% RSLogix 500 project TRIPACK_J.RSS, saved by version 12.00.00.00 %
PROJECT "TRIPACK"    % processor: MicroLogix 1400 %

PROGRAM FILES
  LAD 2   92 rungs
  LAD 3   19 rungs
  LAD 4   43 rungs
  LAD 6   66 rungs
  LAD 18   72 rungs

DATA FILES
  O0 OUTPUT  15 elements
  I1 INPUT  12 elements
  S2 STATUS  66 elements
  B3 BINARY  50 elements
  T4 TIMER  45 elements
  C5 COUNTER  13 elements
  R6 CONTROL  1 elements
  N7 INTEGER  256 elements
  F8 FLOAT  64 elements
  N9   96 elements
  L11   51 elements
  RIX13   13 elements
  RIX14   13 elements
  T15   48 elements
  ST16   18 elements
  RIX17   14 elements
  MG19   11 elements
  MG20   14 elements
  MG22   21 elements

LADDER 2
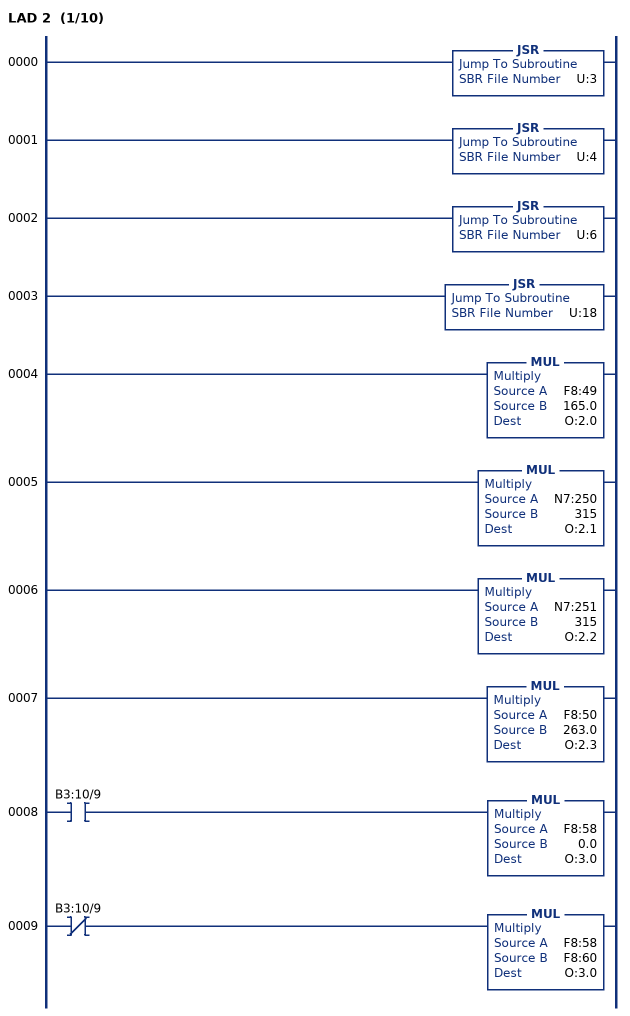
% Rung: 0 %
SOR JSR U:3 EOR
% Rung: 1 %
SOR JSR U:4 EOR
% Rung: 2 %
SOR JSR U:6 EOR
% Rung: 3 %
SOR JSR U:18 EOR
% Rung: 4 %
SOR MUL F8:49 165.0 O:2.0 EOR
% Rung: 5 %
SOR MUL N7:250 315 O:2.1 EOR
% Rung: 6 %
SOR MUL N7:251 315 O:2.2 EOR
% Rung: 7 %
SOR MUL F8:50 263.0 O:2.3 EOR
% Rung: 8 %
SOR XIC B3:10/9 MUL F8:58 0.0 O:3.0 EOR
% Rung: 9 %
SOR XIO B3:10/9 MUL F8:58 F8:60 O:3.0 EOR

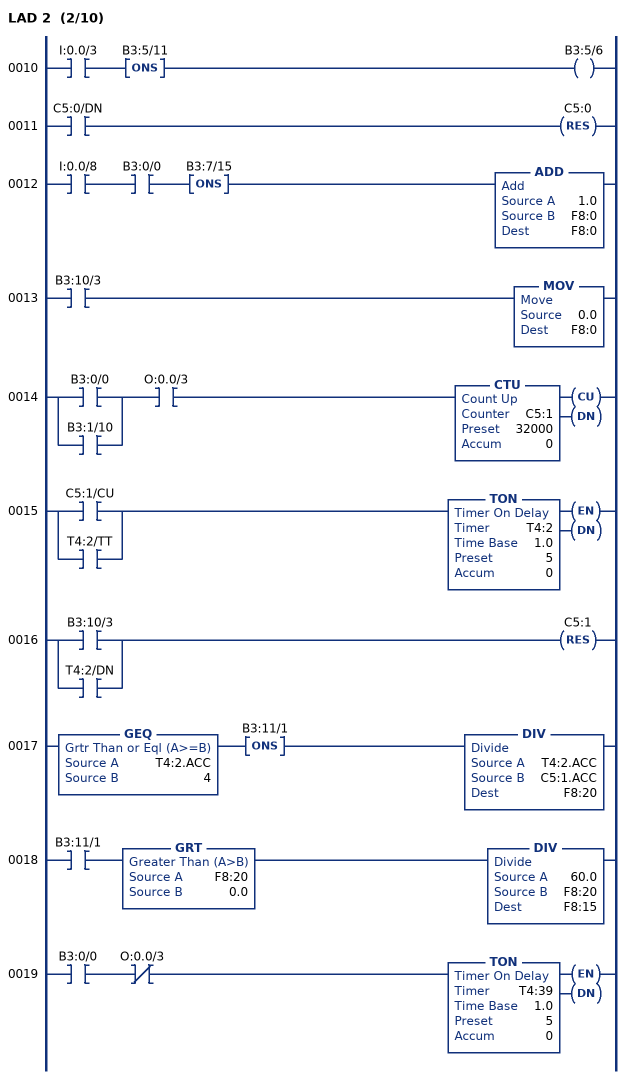
% Rung: 10 %
SOR XIC I:0.0/3 ONS B3:5/11 OTE B3:5/6 EOR
% Rung: 11 %
SOR XIC C5:0/DN RES C5:0 EOR
% Rung: 12 %
SOR XIC I:0.0/8 XIC B3:0/0 ONS B3:7/15 ADD 1.0 F8:0 F8:0 EOR
% Rung: 13 %
SOR XIC B3:10/3 MOV 0.0 F8:0 EOR
% Rung: 14 %
SOR BST XIC B3:0/0 NXB XIC B3:1/10 BND XIC O:0.0/3 CTU C5:1 32000 0 EOR
% Rung: 15 %
SOR BST XIC C5:1/CU NXB XIC T4:2/TT BND TON T4:2 1.0 5 0 EOR
% Rung: 16 %
SOR BST XIC B3:10/3 NXB XIC T4:2/DN BND RES C5:1 EOR
% Rung: 17 %
SOR GEQ T4:2.ACC 4 ONS B3:11/1 DIV T4:2.ACC C5:1.ACC F8:20 EOR
% Rung: 18 %
SOR XIC B3:11/1 GRT F8:20 0.0 DIV 60.0 F8:20 F8:15 EOR
% Rung: 19 %
SOR XIC B3:0/0 XIO O:0.0/3 TON T4:39 1.0 5 0 EOR

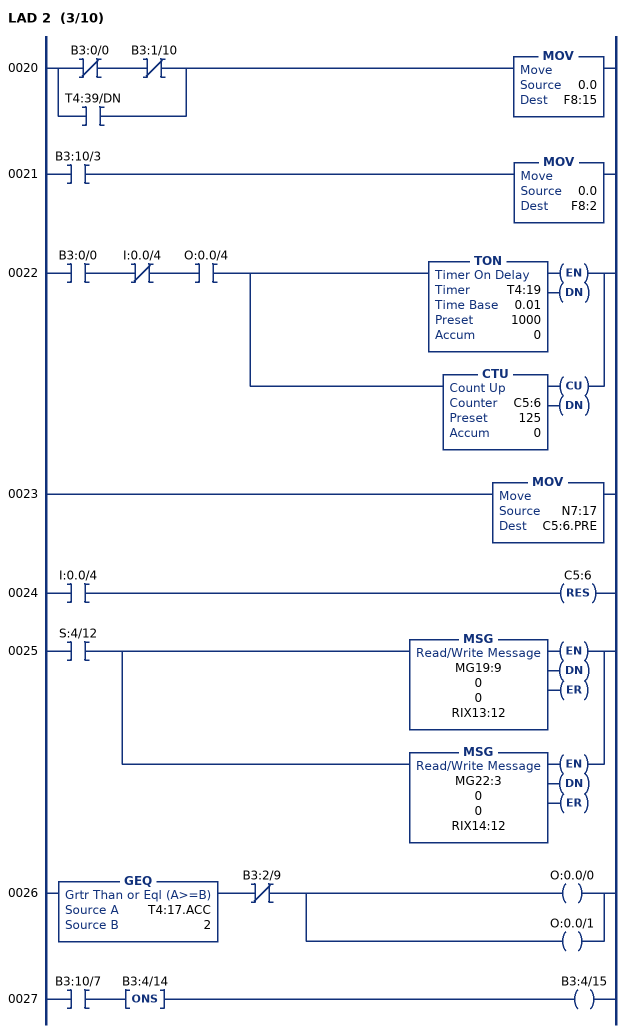
% Rung: 20 %
SOR BST XIO B3:0/0 XIO B3:1/10 NXB XIC T4:39/DN BND MOV 0.0 F8:15 EOR
% Rung: 21 %
SOR XIC B3:10/3 MOV 0.0 F8:2 EOR
% Rung: 22 %
SOR XIC B3:0/0 XIO I:0.0/4 XIC O:0.0/4 BST TON T4:19 0.01 1000 0 NXB CTU C5:6 125 0 BND EOR
% Rung: 23 %
SOR MOV N7:17 C5:6.PRE EOR
% Rung: 24 %
SOR XIC I:0.0/4 RES C5:6 EOR
% Rung: 25 %
SOR XIC S:4/12 BST MSG MG19:9 0 0 RIX13:12 NXB MSG MG22:3 0 0 RIX14:12 BND EOR
%   MSG set-up: CIP Generic | 33 | 0 | ? | 0 | 0 | 0 | 0 | 110.110.110.136:502 | 0 | 0 | 110.110.110.136 | RIX13:12 | E | 884 | 54 | 0 | 374 | 36 | 0 | 0 | 0 %
%   MSG set-up: CIP Generic | 33 | 0 | ? | 0 | 0 | 0 | 0 | 110.110.110.135:502 | 0 | 0 | 110.110.110.135 | RIX14:12 | E | 884 | 54 | 0 | 374 | 36 | 0 | 0 | 0 %
% Rung: 26 %
SOR GEQ T4:17.ACC 2 XIO B3:2/9 BST OTE O:0.0/0 NXB OTE O:0.0/1 BND EOR
% Rung: 27 %
SOR XIC B3:10/7 ONS B3:4/14 OTE B3:4/15 EOR

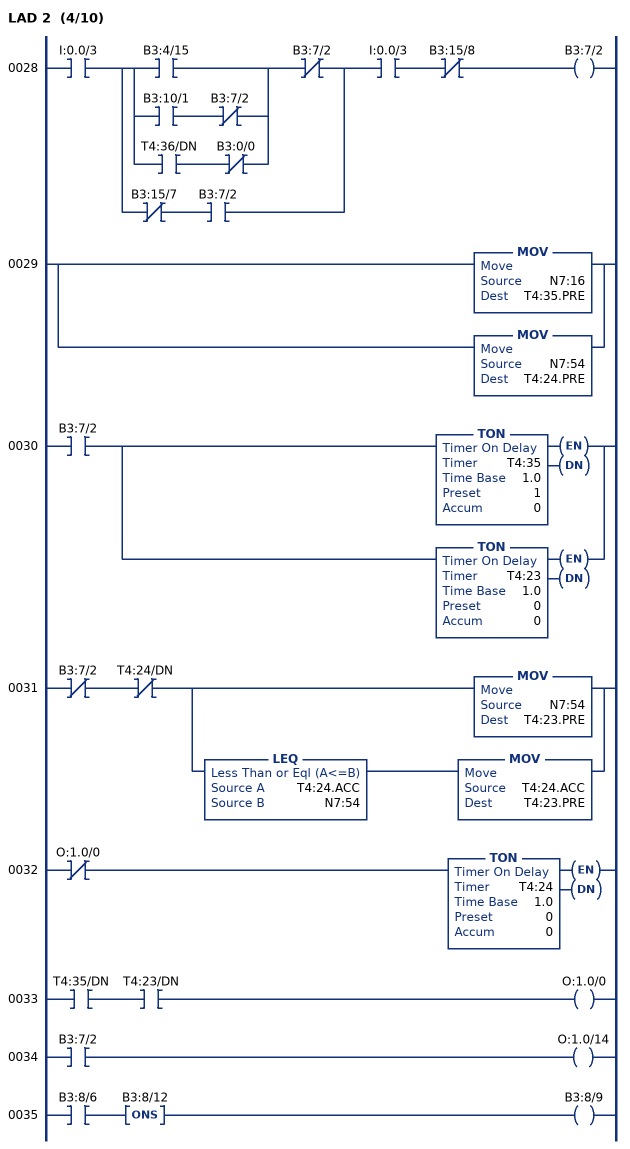
% Rung: 28 %
SOR XIC I:0.0/3 BST BST XIC B3:4/15 NXB XIC B3:10/1 XIO B3:7/2 NXB XIC T4:36/DN XIO B3:0/0 BND XIO B3:7/2 NXB XIO B3:15/7 XIC B3:7/2 BND XIC I:0.0/3 XIO B3:15/8 OTE B3:7/2 EOR
% Rung: 29 %
SOR BST MOV N7:16 T4:35.PRE NXB MOV N7:54 T4:24.PRE BND EOR
% Rung: 30 %
SOR XIC B3:7/2 BST TON T4:35 1.0 1 0 NXB TON T4:23 1.0 0 0 BND EOR
% Rung: 31 %
SOR XIO B3:7/2 XIO T4:24/DN BST MOV N7:54 T4:23.PRE NXB LEQ T4:24.ACC N7:54 MOV T4:24.ACC T4:23.PRE BND EOR
% Rung: 32 %
SOR XIO O:1.0/0 TON T4:24 1.0 0 0 EOR
% Rung: 33 %
SOR XIC T4:35/DN XIC T4:23/DN OTE O:1.0/0 EOR
% Rung: 34 %
SOR XIC B3:7/2 OTE O:1.0/14 EOR
% Rung: 35 %
SOR XIC B3:8/6 ONS B3:8/12 OTE B3:8/9 EOR

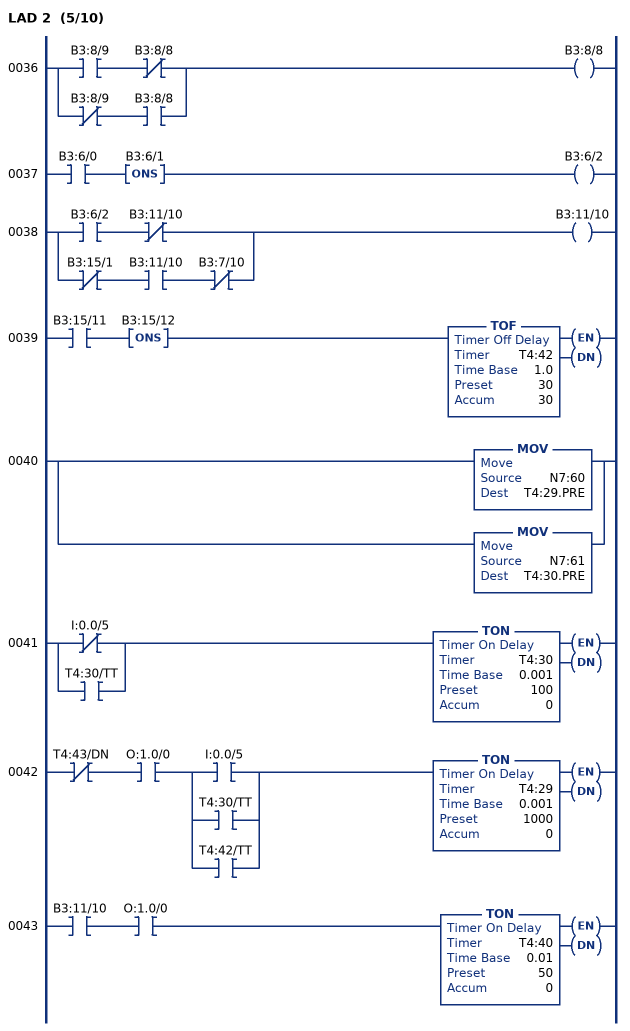
% Rung: 36 %
SOR BST XIC B3:8/9 XIO B3:8/8 NXB XIO B3:8/9 XIC B3:8/8 BND OTE B3:8/8 EOR
% Rung: 37 %
SOR XIC B3:6/0 ONS B3:6/1 OTE B3:6/2 EOR
% Rung: 38 %
SOR BST XIC B3:6/2 XIO B3:11/10 NXB XIO B3:15/1 XIC B3:11/10 XIO B3:7/10 BND OTE B3:11/10 EOR
% Rung: 39 %
SOR XIC B3:15/11 ONS B3:15/12 TOF T4:42 1.0 30 30 EOR
% Rung: 40 %
SOR BST MOV N7:60 T4:29.PRE NXB MOV N7:61 T4:30.PRE BND EOR
% Rung: 41 %
SOR BST XIO I:0.0/5 NXB XIC T4:30/TT BND TON T4:30 0.001 100 0 EOR
% Rung: 42 %
SOR XIO T4:43/DN XIC O:1.0/0 BST XIC I:0.0/5 NXB XIC T4:30/TT NXB XIC T4:42/TT BND TON T4:29 0.001 1000 0 EOR
% Rung: 43 %
SOR XIC B3:11/10 XIC O:1.0/0 TON T4:40 0.01 50 0 EOR

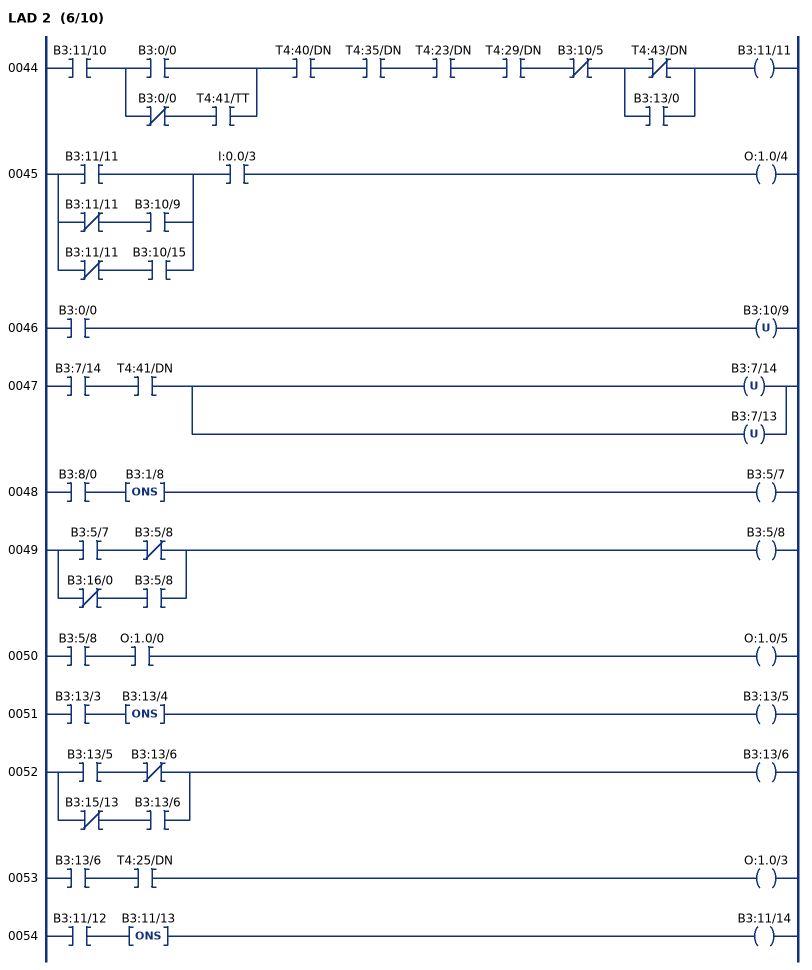
% Rung: 44 %
SOR XIC B3:11/10 BST XIC B3:0/0 NXB XIO B3:0/0 XIC T4:41/TT BND XIC T4:40/DN XIC T4:35/DN XIC T4:23/DN XIC T4:29/DN XIO B3:10/5 BST XIO T4:43/DN NXB XIC B3:13/0 BND OTE B3:11/11 EOR
% Rung: 45 %
SOR BST XIC B3:11/11 NXB XIO B3:11/11 XIC B3:10/9 NXB XIO B3:11/11 XIC B3:10/15 BND XIC I:0.0/3 OTE O:1.0/4 EOR
% Rung: 46 %
SOR XIC B3:0/0 OTU B3:10/9 EOR
% Rung: 47 %
SOR XIC B3:7/14 XIC T4:41/DN BST OTU B3:7/14 NXB OTU B3:7/13 BND EOR
% Rung: 48 %
SOR XIC B3:8/0 ONS B3:1/8 OTE B3:5/7 EOR
% Rung: 49 %
SOR BST XIC B3:5/7 XIO B3:5/8 NXB XIO B3:16/0 XIC B3:5/8 BND OTE B3:5/8 EOR
% Rung: 50 %
SOR XIC B3:5/8 XIC O:1.0/0 OTE O:1.0/5 EOR
% Rung: 51 %
SOR XIC B3:13/3 ONS B3:13/4 OTE B3:13/5 EOR
% Rung: 52 %
SOR BST XIC B3:13/5 XIO B3:13/6 NXB XIO B3:15/13 XIC B3:13/6 BND OTE B3:13/6 EOR
% Rung: 53 %
SOR XIC B3:13/6 XIC T4:25/DN OTE O:1.0/3 EOR
% Rung: 54 %
SOR XIC B3:11/12 ONS B3:11/13 OTE B3:11/14 EOR

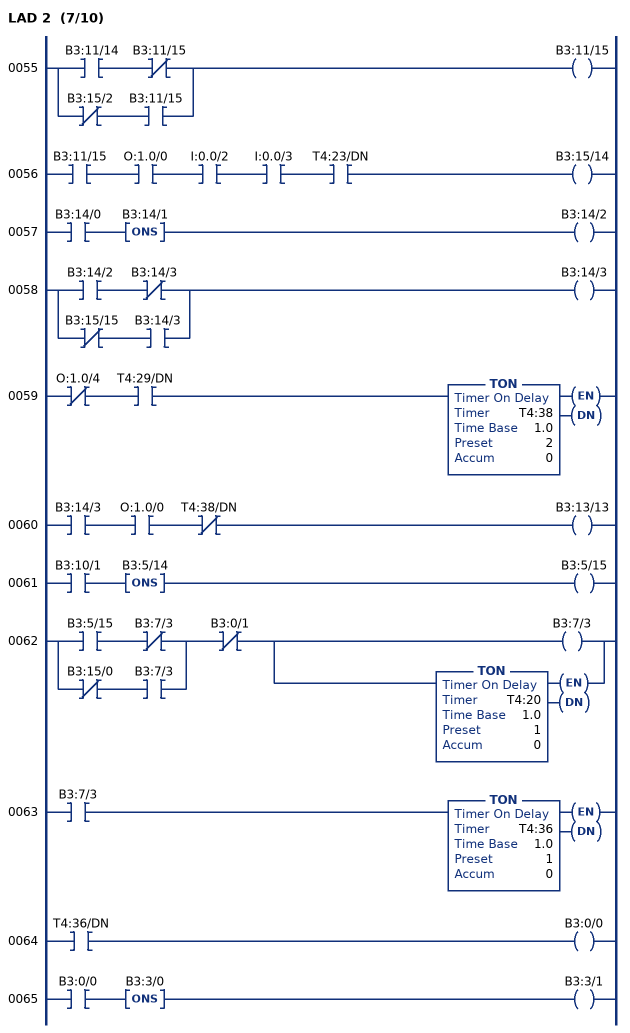
% Rung: 55 %
SOR BST XIC B3:11/14 XIO B3:11/15 NXB XIO B3:15/2 XIC B3:11/15 BND OTE B3:11/15 EOR
% Rung: 56 %
SOR XIC B3:11/15 XIC O:1.0/0 XIC I:0.0/2 XIC I:0.0/3 XIC T4:23/DN OTE B3:15/14 EOR
% Rung: 57 %
SOR XIC B3:14/0 ONS B3:14/1 OTE B3:14/2 EOR
% Rung: 58 %
SOR BST XIC B3:14/2 XIO B3:14/3 NXB XIO B3:15/15 XIC B3:14/3 BND OTE B3:14/3 EOR
% Rung: 59 %
SOR XIO O:1.0/4 XIC T4:29/DN TON T4:38 1.0 2 0 EOR
% Rung: 60 %
SOR XIC B3:14/3 XIC O:1.0/0 XIO T4:38/DN OTE B3:13/13 EOR
% Rung: 61 %
SOR XIC B3:10/1 ONS B3:5/14 OTE B3:5/15 EOR
% Rung: 62 %
SOR BST XIC B3:5/15 XIO B3:7/3 NXB XIO B3:15/0 XIC B3:7/3 BND XIO B3:0/1 BST OTE B3:7/3 NXB TON T4:20 1.0 1 0 BND EOR
% Rung: 63 %
SOR XIC B3:7/3 TON T4:36 1.0 1 0 EOR
% Rung: 64 %
SOR XIC T4:36/DN OTE B3:0/0 EOR
% Rung: 65 %
SOR XIC B3:0/0 ONS B3:3/0 OTE B3:3/1 EOR

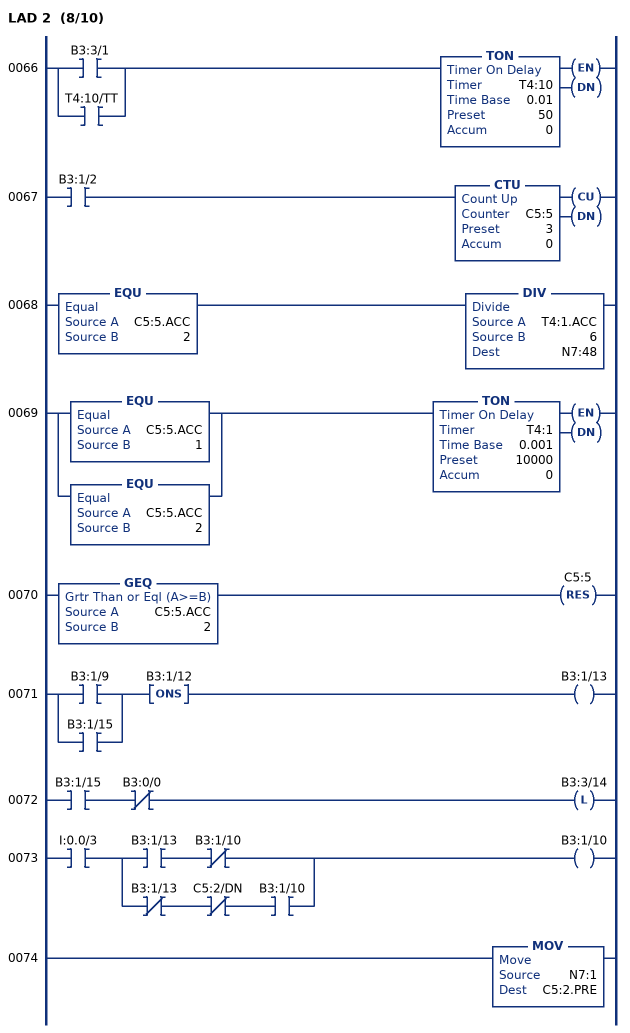
% Rung: 66 %
SOR BST XIC B3:3/1 NXB XIC T4:10/TT BND TON T4:10 0.01 50 0 EOR
% Rung: 67 %
SOR XIC B3:1/2 CTU C5:5 3 0 EOR
% Rung: 68 %
SOR EQU C5:5.ACC 2 DIV T4:1.ACC 6 N7:48 EOR
% Rung: 69 %
SOR BST EQU C5:5.ACC 1 NXB EQU C5:5.ACC 2 BND TON T4:1 0.001 10000 0 EOR
% Rung: 70 %
SOR GEQ C5:5.ACC 2 RES C5:5 EOR
% Rung: 71 %
SOR BST XIC B3:1/9 NXB XIC B3:1/15 BND ONS B3:1/12 OTE B3:1/13 EOR
% Rung: 72 %
SOR XIC B3:1/15 XIO B3:0/0 OTL B3:3/14 EOR
% Rung: 73 %
SOR XIC I:0.0/3 BST XIC B3:1/13 XIO B3:1/10 NXB XIO B3:1/13 XIO C5:2/DN XIC B3:1/10 BND OTE B3:1/10 EOR
% Rung: 74 %
SOR MOV N7:1 C5:2.PRE EOR

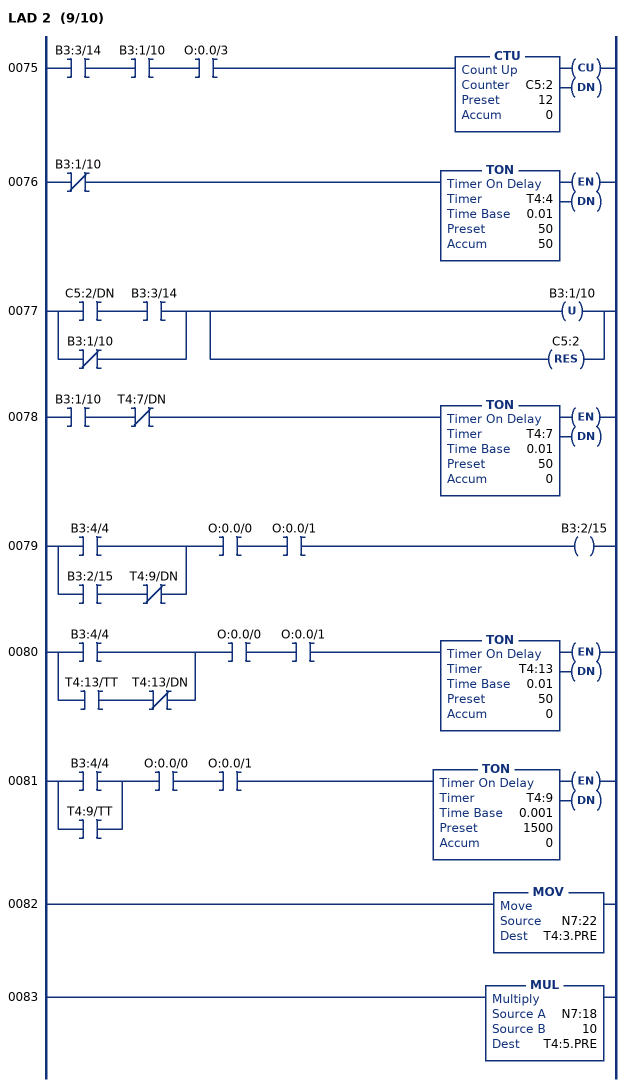
% Rung: 75 %
SOR XIC B3:3/14 XIC B3:1/10 XIC O:0.0/3 CTU C5:2 12 0 EOR
% Rung: 76 %
SOR XIO B3:1/10 TON T4:4 0.01 50 50 EOR
% Rung: 77 %
SOR BST XIC C5:2/DN XIC B3:3/14 NXB XIO B3:1/10 BND BST OTU B3:1/10 NXB RES C5:2 BND EOR
% Rung: 78 %
SOR XIC B3:1/10 XIO T4:7/DN TON T4:7 0.01 50 0 EOR
% Rung: 79 %
SOR BST XIC B3:4/4 NXB XIC B3:2/15 XIO T4:9/DN BND XIC O:0.0/0 XIC O:0.0/1 OTE B3:2/15 EOR
% Rung: 80 %
SOR BST XIC B3:4/4 NXB XIC T4:13/TT XIO T4:13/DN BND XIC O:0.0/0 XIC O:0.0/1 TON T4:13 0.01 50 0 EOR
% Rung: 81 %
SOR BST XIC B3:4/4 NXB XIC T4:9/TT BND XIC O:0.0/0 XIC O:0.0/1 TON T4:9 0.001 1500 0 EOR
% Rung: 82 %
SOR MOV N7:22 T4:3.PRE EOR
% Rung: 83 %
SOR MUL N7:18 10 T4:5.PRE EOR

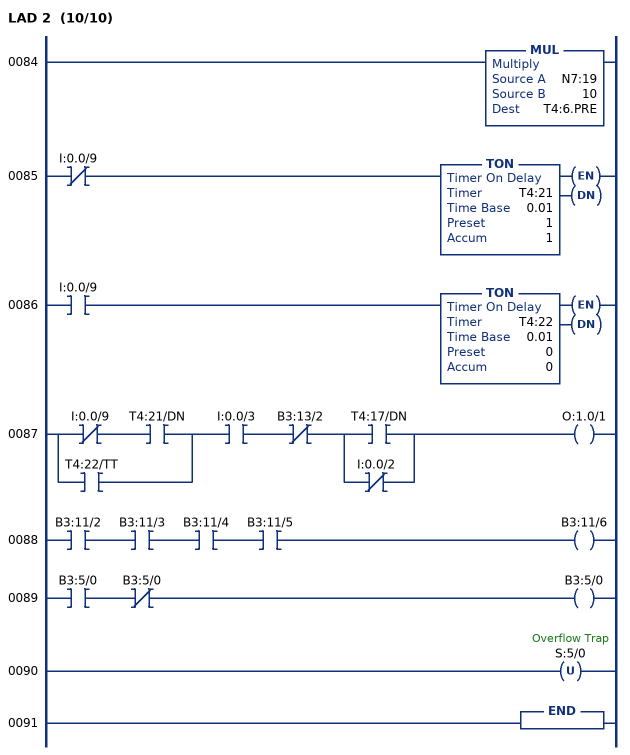
% Rung: 84 %
SOR MUL N7:19 10 T4:6.PRE EOR
% Rung: 85 %
SOR XIO I:0.0/9 TON T4:21 0.01 1 1 EOR
% Rung: 86 %
SOR XIC I:0.0/9 TON T4:22 0.01 0 0 EOR
% Rung: 87 %
SOR BST XIO I:0.0/9 XIC T4:21/DN NXB XIC T4:22/TT BND XIC I:0.0/3 XIO B3:13/2 BST XIC T4:17/DN NXB XIO I:0.0/2 BND OTE O:1.0/1 EOR
% Rung: 88 %
SOR XIC B3:11/2 XIC B3:11/3 XIC B3:11/4 XIC B3:11/5 OTE B3:11/6 EOR
% Rung: 89 %
SOR XIC B3:5/0 XIO B3:5/0 OTE B3:5/0 EOR
% Rung: 90 %
SOR OTU S:5/0 EOR
%   S:5/0  "Overflow Trap" %
% Rung: 91 %
SOR END EOR

LADDER 3
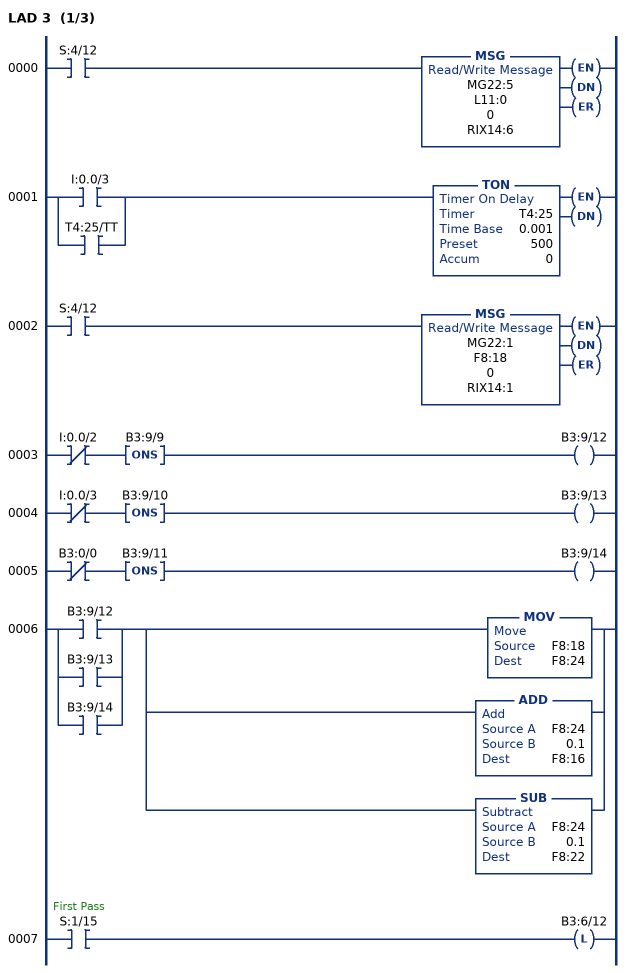
% Rung: 0 %
SOR XIC S:4/12 MSG MG22:5 L11:0 0 RIX14:6 EOR
%   MSG set-up: CIP Generic | 33 | 64 | ? | L11:0 | 0 | 0 | 0 | 110.110.110.135:502 | 0 | 0 | 110.110.110.135 | RIX14:6 | E | 4 | 113 | 3 | 4 | 71 | 3 | 0 | 0 %
% Rung: 1 %
SOR BST XIC I:0.0/3 NXB XIC T4:25/TT BND TON T4:25 0.001 500 0 EOR
% Rung: 2 %
SOR XIC S:4/12 MSG MG22:1 F8:18 0 RIX14:1 EOR
%   MSG set-up: CIP Generic | 33 | 4 | ? | F8:18 | 0 | 0 | 0 | 110.110.110.135:502 | 0 | 0 | 110.110.110.135 | RIX14:1 | E | 884 | 210 | 2 | 374 | D2 | 2 | 0 | 0 %
% Rung: 3 %
SOR XIO I:0.0/2 ONS B3:9/9 OTE B3:9/12 EOR
% Rung: 4 %
SOR XIO I:0.0/3 ONS B3:9/10 OTE B3:9/13 EOR
% Rung: 5 %
SOR XIO B3:0/0 ONS B3:9/11 OTE B3:9/14 EOR
% Rung: 6 %
SOR BST XIC B3:9/12 NXB XIC B3:9/13 NXB XIC B3:9/14 BND BST MOV F8:18 F8:24 NXB ADD F8:24 0.1 F8:16 NXB SUB F8:24 0.1 F8:22 BND EOR
% Rung: 7 %
SOR XIC S:1/15 OTL B3:6/12 EOR
%   S:1/15  "First Pass" %

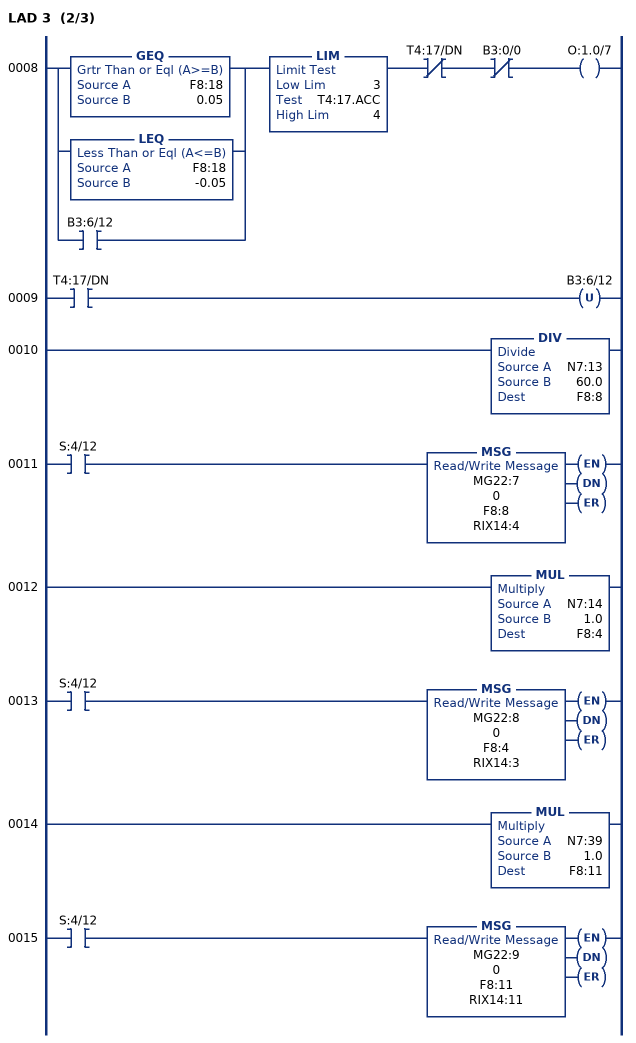
% Rung: 8 %
SOR BST BST GEQ F8:18 0.05 NXB LEQ F8:18 -0.05 BND NXB XIC B3:6/12 BND LIM 3 T4:17.ACC 4 XIO T4:17/DN XIO B3:0/0 OTE O:1.0/7 EOR
% Rung: 9 %
SOR XIC T4:17/DN OTU B3:6/12 EOR
% Rung: 10 %
SOR DIV N7:13 60.0 F8:8 EOR
% Rung: 11 %
SOR XIC S:4/12 MSG MG22:7 0 F8:8 RIX14:4 EOR
%   MSG set-up: CIP Generic | 33 | 0 | ? | 0 | 0 | 0 | 0 | 110.110.110.135:502 | 0 | 0 | 110.110.110.135 | RIX14:4 | 10 | 884 | 278 | 2 | 374 | 116 | 2 | 4 | F8:8 %
% Rung: 12 %
SOR MUL N7:14 1.0 F8:4 EOR
% Rung: 13 %
SOR XIC S:4/12 MSG MG22:8 0 F8:4 RIX14:3 EOR
%   MSG set-up: CIP Generic | 33 | 0 | ? | 0 | 0 | 0 | 0 | 110.110.110.135:502 | 0 | 0 | 110.110.110.135 | RIX14:3 | 10 | 884 | 279 | 2 | 374 | 117 | 2 | 4 | F8:4 %
% Rung: 14 %
SOR MUL N7:39 1.0 F8:11 EOR
% Rung: 15 %
SOR XIC S:4/12 MSG MG22:9 0 F8:11 RIX14:11 EOR
%   MSG set-up: CIP Generic | 33 | 0 | ? | 0 | 0 | 0 | 0 | 110.110.110.135:502 | 0 | 0 | 110.110.110.135 | RIX14:11 | 10 | 884 | 280 | 2 | 374 | 118 | 2 | 4 | F8:11 %

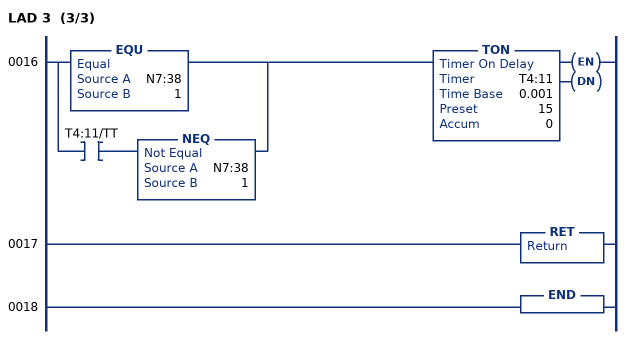
% Rung: 16 %
SOR BST EQU N7:38 1 NXB XIC T4:11/TT NEQ N7:38 1 BND TON T4:11 0.001 15 0 EOR
% Rung: 17 %
SOR RET EOR
% Rung: 18 %
SOR END EOR

LADDER 4
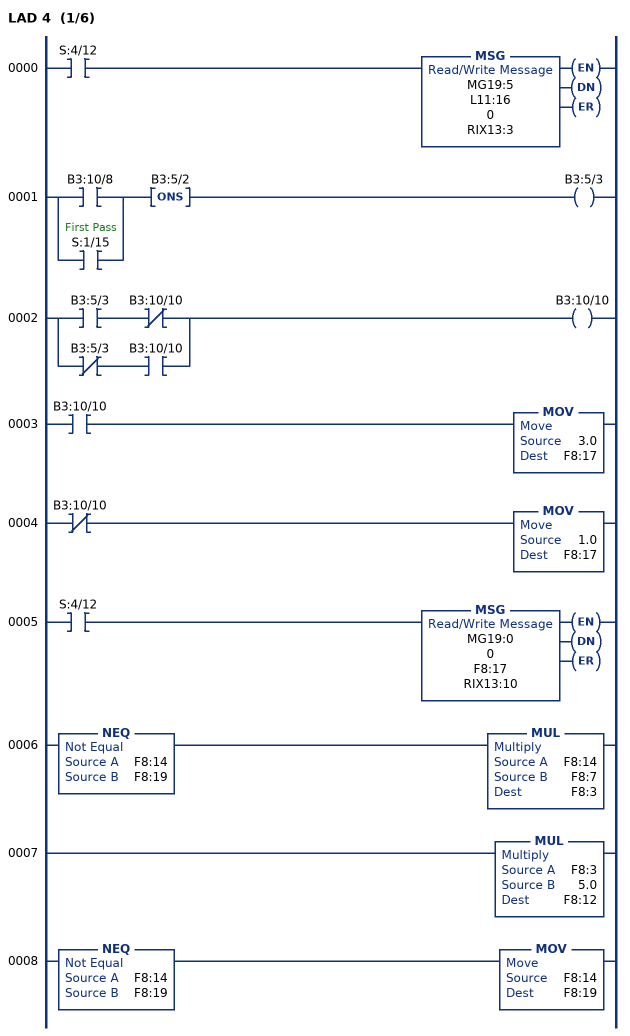
% Rung: 0 %
SOR XIC S:4/12 MSG MG19:5 L11:16 0 RIX13:3 EOR
%   MSG set-up: CIP Generic | 33 | 64 | ? | L11:16 | 0 | 0 | 0 | 110.110.110.136:502 | 0 | 0 | 110.110.110.136 | RIX13:3 | E | 4 | 113 | 3 | 4 | 71 | 3 | 0 | 0 %
% Rung: 1 %
SOR BST XIC B3:10/8 NXB XIC S:1/15 BND ONS B3:5/2 OTE B3:5/3 EOR
%   S:1/15  "First Pass" %
% Rung: 2 %
SOR BST XIC B3:5/3 XIO B3:10/10 NXB XIO B3:5/3 XIC B3:10/10 BND OTE B3:10/10 EOR
% Rung: 3 %
SOR XIC B3:10/10 MOV 3.0 F8:17 EOR
% Rung: 4 %
SOR XIO B3:10/10 MOV 1.0 F8:17 EOR
% Rung: 5 %
SOR XIC S:4/12 MSG MG19:0 0 F8:17 RIX13:10 EOR
%   MSG set-up: CIP Generic | 33 | 0 | ? | 0 | 0 | 0 | 0 | 110.110.110.136:502 | 0 | 0 | 110.110.110.136 | RIX13:10 | 10 | 884 | 272 | 2 | 374 | 110 | 2 | 4 | F8:17 %
% Rung: 6 %
SOR NEQ F8:14 F8:19 MUL F8:14 F8:7 F8:3 EOR
% Rung: 7 %
SOR MUL F8:3 5.0 F8:12 EOR
% Rung: 8 %
SOR NEQ F8:14 F8:19 MOV F8:14 F8:19 EOR

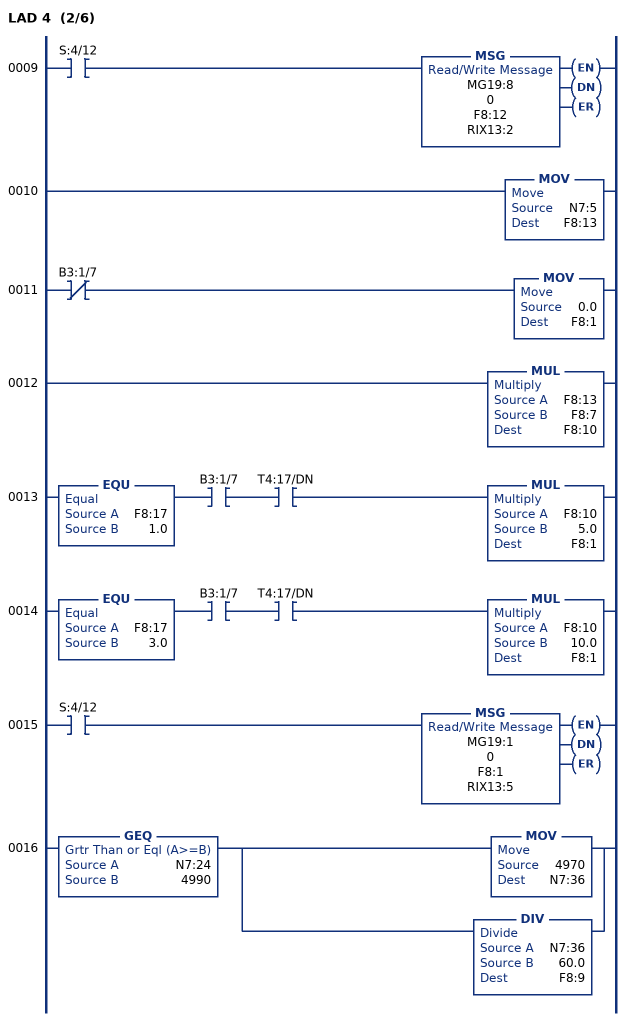
% Rung: 9 %
SOR XIC S:4/12 MSG MG19:8 0 F8:12 RIX13:2 EOR
%   MSG set-up: CIP Generic | 33 | 0 | ? | 0 | 0 | 0 | 0 | 110.110.110.136:502 | 0 | 0 | 110.110.110.136 | RIX13:2 | 10 | 884 | 275 | 2 | 374 | 113 | 2 | 4 | F8:12 %
% Rung: 10 %
SOR MOV N7:5 F8:13 EOR
% Rung: 11 %
SOR XIO B3:1/7 MOV 0.0 F8:1 EOR
% Rung: 12 %
SOR MUL F8:13 F8:7 F8:10 EOR
% Rung: 13 %
SOR EQU F8:17 1.0 XIC B3:1/7 XIC T4:17/DN MUL F8:10 5.0 F8:1 EOR
% Rung: 14 %
SOR EQU F8:17 3.0 XIC B3:1/7 XIC T4:17/DN MUL F8:10 10.0 F8:1 EOR
% Rung: 15 %
SOR XIC S:4/12 MSG MG19:1 0 F8:1 RIX13:5 EOR
%   MSG set-up: CIP Generic | 33 | 0 | ? | 0 | 0 | 0 | 0 | 110.110.110.136:502 | 0 | 0 | 110.110.110.136 | RIX13:5 | 10 | 884 | 274 | 2 | 374 | 112 | 2 | 4 | F8:1 %
% Rung: 16 %
SOR GEQ N7:24 4990 BST MOV 4970 N7:36 NXB DIV N7:36 60.0 F8:9 BND EOR

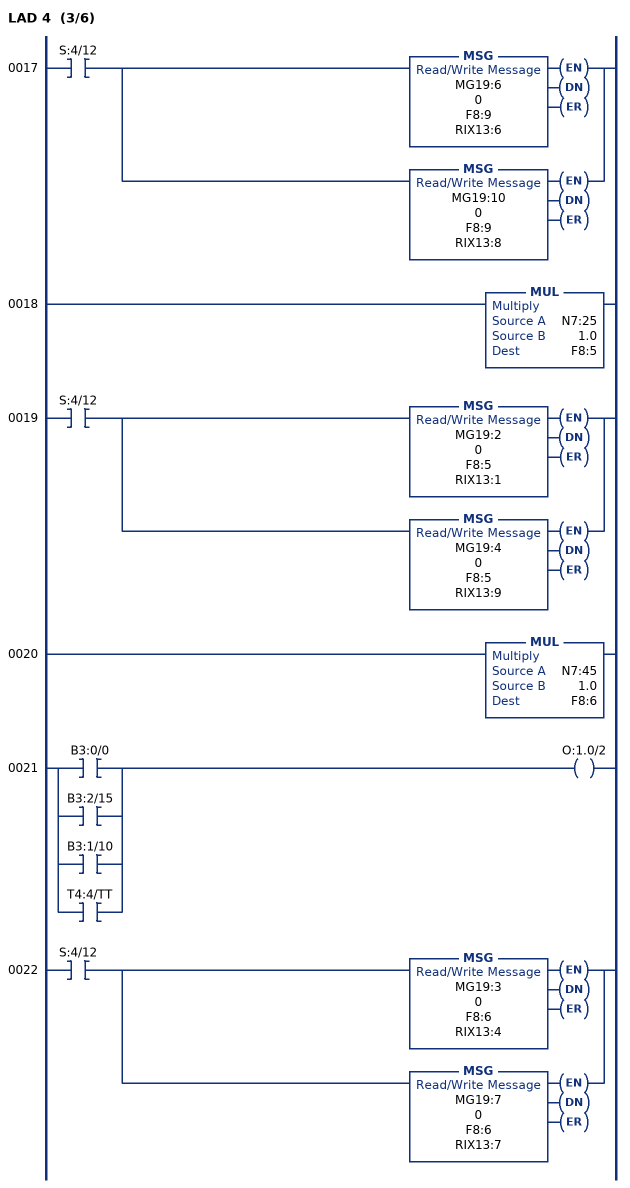
% Rung: 17 %
SOR XIC S:4/12 BST MSG MG19:6 0 F8:9 RIX13:6 NXB MSG MG19:10 0 F8:9 RIX13:8 BND EOR
%   MSG set-up: CIP Generic | 33 | 0 | ? | 0 | 0 | 0 | 0 | 110.110.110.136:502 | 0 | 0 | 110.110.110.136 | RIX13:6 | 10 | 884 | 278 | 2 | 374 | 116 | 2 | 4 | F8:9 %
%   MSG set-up: CIP Generic | 33 | 0 | ? | 0 | 0 | 0 | 0 | 110.110.110.136:502 | 0 | 0 | 110.110.110.136 | RIX13:8 | 10 | 884 | 289 | 2 | 374 | 121 | 2 | 1 | F8:9 %
% Rung: 18 %
SOR MUL N7:25 1.0 F8:5 EOR
% Rung: 19 %
SOR XIC S:4/12 BST MSG MG19:2 0 F8:5 RIX13:1 NXB MSG MG19:4 0 F8:5 RIX13:9 BND EOR
%   MSG set-up: CIP Generic | 33 | 0 | ? | 0 | 0 | 0 | 0 | 110.110.110.136:502 | 0 | 0 | 110.110.110.136 | RIX13:1 | 10 | 884 | 279 | 2 | 374 | 117 | 2 | 4 | F8:5 %
%   MSG set-up: CIP Generic | 33 | 0 | ? | 0 | 0 | 0 | 0 | 110.110.110.136:502 | 0 | 0 | 110.110.110.136 | RIX13:9 | 10 | 884 | 290 | 2 | 374 | 122 | 2 | 4 | F8:5 %
% Rung: 20 %
SOR MUL N7:45 1.0 F8:6 EOR
% Rung: 21 %
SOR BST XIC B3:0/0 NXB XIC B3:2/15 NXB XIC B3:1/10 NXB XIC T4:4/TT BND OTE O:1.0/2 EOR
% Rung: 22 %
SOR XIC S:4/12 BST MSG MG19:3 0 F8:6 RIX13:4 NXB MSG MG19:7 0 F8:6 RIX13:7 BND EOR
%   MSG set-up: CIP Generic | 33 | 0 | ? | 0 | 0 | 0 | 0 | 110.110.110.136:502 | 0 | 0 | 110.110.110.136 | RIX13:4 | 10 | 884 | 280 | 2 | 374 | 118 | 2 | 4 | F8:6 %
%   MSG set-up: CIP Generic | 33 | 0 | ? | 0 | 0 | 0 | 0 | 110.110.110.136:502 | 0 | 0 | 110.110.110.136 | RIX13:7 | 10 | 884 | 291 | 2 | 374 | 123 | 2 | 1 | F8:6 %

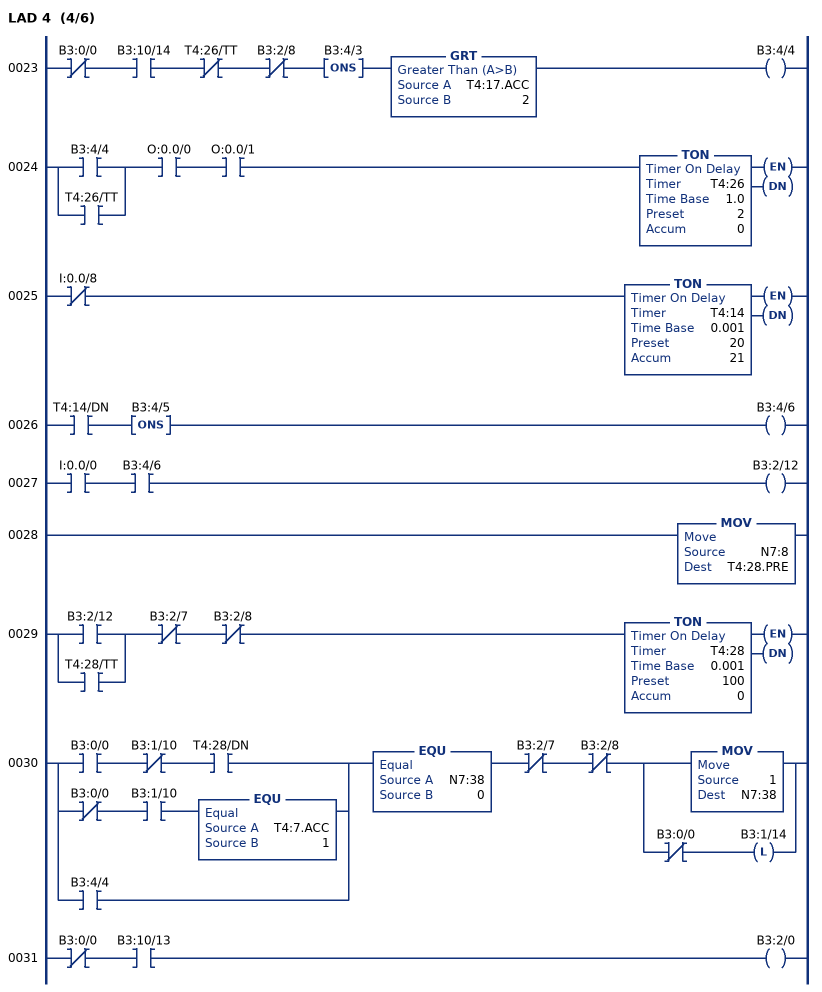
% Rung: 23 %
SOR XIO B3:0/0 XIC B3:10/14 XIO T4:26/TT XIO B3:2/8 ONS B3:4/3 GRT T4:17.ACC 2 OTE B3:4/4 EOR
% Rung: 24 %
SOR BST XIC B3:4/4 NXB XIC T4:26/TT BND XIC O:0.0/0 XIC O:0.0/1 TON T4:26 1.0 2 0 EOR
% Rung: 25 %
SOR XIO I:0.0/8 TON T4:14 0.001 20 21 EOR
% Rung: 26 %
SOR XIC T4:14/DN ONS B3:4/5 OTE B3:4/6 EOR
% Rung: 27 %
SOR XIC I:0.0/0 XIC B3:4/6 OTE B3:2/12 EOR
% Rung: 28 %
SOR MOV N7:8 T4:28.PRE EOR
% Rung: 29 %
SOR BST XIC B3:2/12 NXB XIC T4:28/TT BND XIO B3:2/7 XIO B3:2/8 TON T4:28 0.001 100 0 EOR
% Rung: 30 %
SOR BST BST XIC B3:0/0 XIO B3:1/10 XIC T4:28/DN NXB XIO B3:0/0 XIC B3:1/10 EQU T4:7.ACC 1 BND NXB XIC B3:4/4 BND EQU N7:38 0 XIO B3:2/7 XIO B3:2/8 BST MOV 1 N7:38 NXB XIO B3:0/0 OTL B3:1/14 BND EOR
% Rung: 31 %
SOR XIO B3:0/0 XIC B3:10/13 OTE B3:2/0 EOR

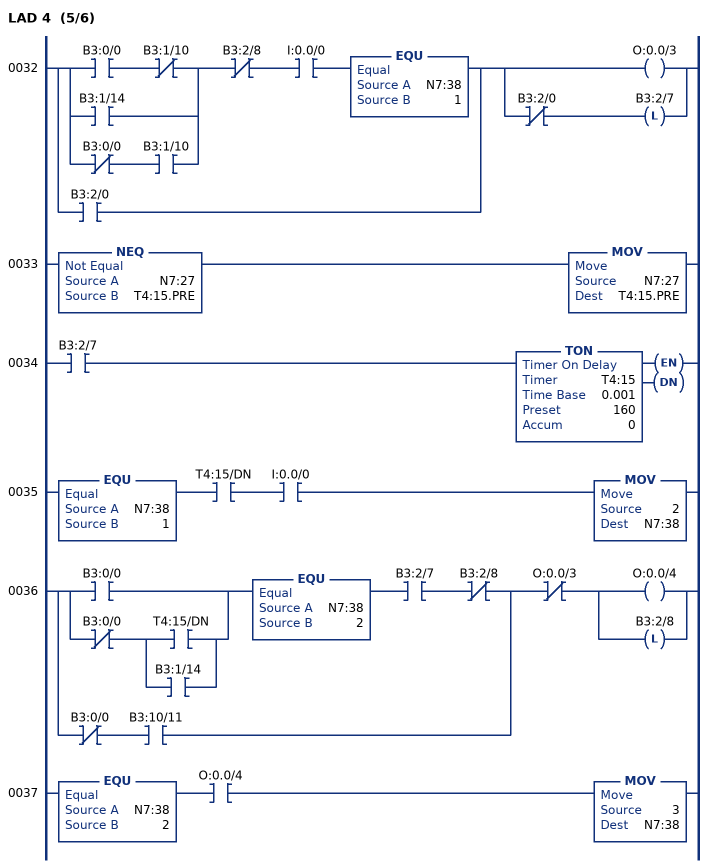
% Rung: 32 %
SOR BST BST XIC B3:0/0 XIO B3:1/10 NXB XIC B3:1/14 NXB XIO B3:0/0 XIC B3:1/10 BND XIO B3:2/8 XIC I:0.0/0 EQU N7:38 1 NXB XIC B3:2/0 BND BST OTE O:0.0/3 NXB XIO B3:2/0 OTL B3:2/7 BND EOR
% Rung: 33 %
SOR NEQ N7:27 T4:15.PRE MOV N7:27 T4:15.PRE EOR
% Rung: 34 %
SOR XIC B3:2/7 TON T4:15 0.001 160 0 EOR
% Rung: 35 %
SOR EQU N7:38 1 XIC T4:15/DN XIC I:0.0/0 MOV 2 N7:38 EOR
% Rung: 36 %
SOR BST BST XIC B3:0/0 NXB XIO B3:0/0 BST XIC T4:15/DN NXB XIC B3:1/14 BND BND EQU N7:38 2 XIC B3:2/7 XIO B3:2/8 NXB XIO B3:0/0 XIC B3:10/11 BND XIO O:0.0/3 BST OTE O:0.0/4 NXB OTL B3:2/8 BND EOR
% Rung: 37 %
SOR EQU N7:38 2 XIC O:0.0/4 MOV 3 N7:38 EOR

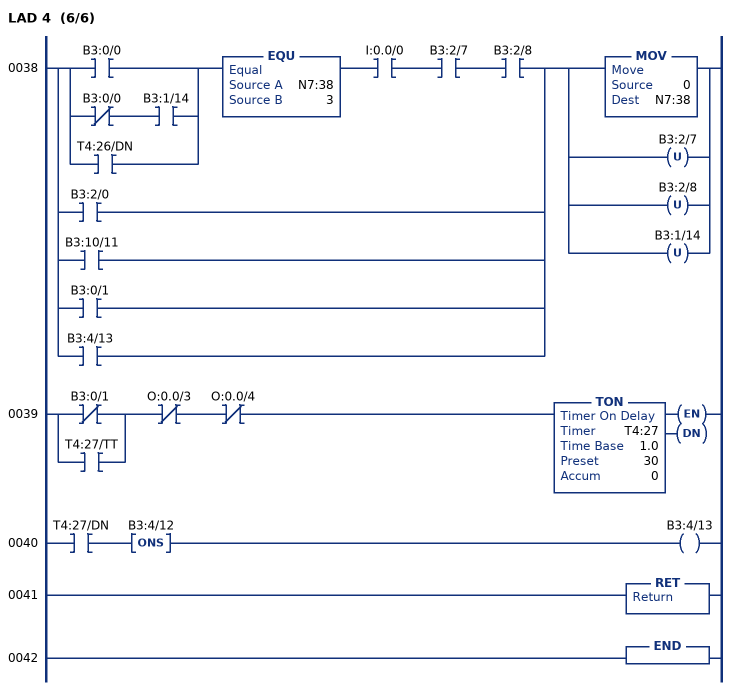
% Rung: 38 %
SOR BST BST XIC B3:0/0 NXB XIO B3:0/0 XIC B3:1/14 NXB XIC T4:26/DN BND EQU N7:38 3 XIC I:0.0/0 XIC B3:2/7 XIC B3:2/8 NXB XIC B3:2/0 NXB XIC B3:10/11 NXB XIC B3:0/1 NXB XIC B3:4/13 BND BST MOV 0 N7:38 NXB OTU B3:2/7 NXB OTU B3:2/8 NXB OTU B3:1/14 BND EOR
% Rung: 39 %
SOR BST XIO B3:0/1 NXB XIC T4:27/TT BND XIO O:0.0/3 XIO O:0.0/4 TON T4:27 1.0 30 0 EOR
% Rung: 40 %
SOR XIC T4:27/DN ONS B3:4/12 OTE B3:4/13 EOR
% Rung: 41 %
SOR RET EOR
% Rung: 42 %
SOR END EOR

LADDER 6
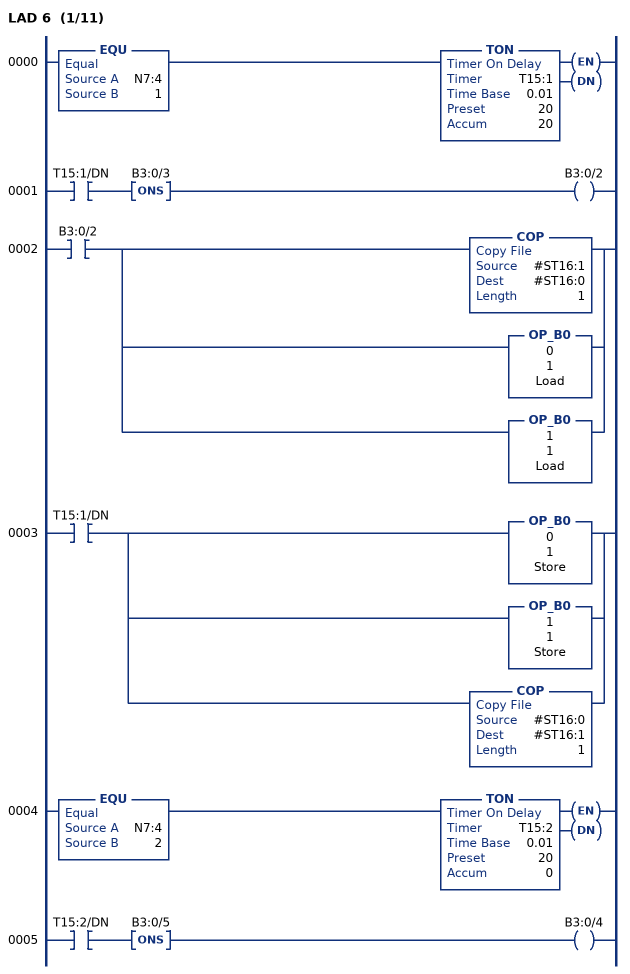
% Rung: 0 %
SOR EQU N7:4 1 TON T15:1 0.01 20 20 EOR
% Rung: 1 %
SOR XIC T15:1/DN ONS B3:0/3 OTE B3:0/2 EOR
% Rung: 2 %
SOR XIC B3:0/2 BST COP #ST16:1 #ST16:0 1 NXB OP_B0 0 1 Load NXB OP_B0 1 1 Load BND EOR
% Rung: 3 %
SOR XIC T15:1/DN BST OP_B0 0 1 Store NXB OP_B0 1 1 Store NXB COP #ST16:0 #ST16:1 1 BND EOR
% Rung: 4 %
SOR EQU N7:4 2 TON T15:2 0.01 20 0 EOR
% Rung: 5 %
SOR XIC T15:2/DN ONS B3:0/5 OTE B3:0/4 EOR

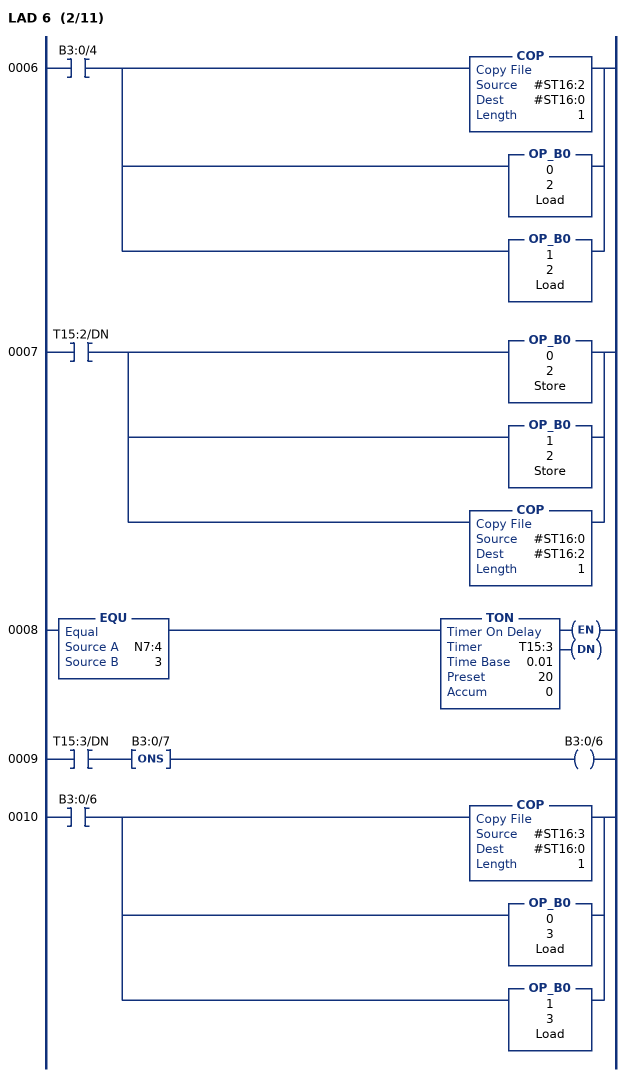
% Rung: 6 %
SOR XIC B3:0/4 BST COP #ST16:2 #ST16:0 1 NXB OP_B0 0 2 Load NXB OP_B0 1 2 Load BND EOR
% Rung: 7 %
SOR XIC T15:2/DN BST OP_B0 0 2 Store NXB OP_B0 1 2 Store NXB COP #ST16:0 #ST16:2 1 BND EOR
% Rung: 8 %
SOR EQU N7:4 3 TON T15:3 0.01 20 0 EOR
% Rung: 9 %
SOR XIC T15:3/DN ONS B3:0/7 OTE B3:0/6 EOR
% Rung: 10 %
SOR XIC B3:0/6 BST COP #ST16:3 #ST16:0 1 NXB OP_B0 0 3 Load NXB OP_B0 1 3 Load BND EOR

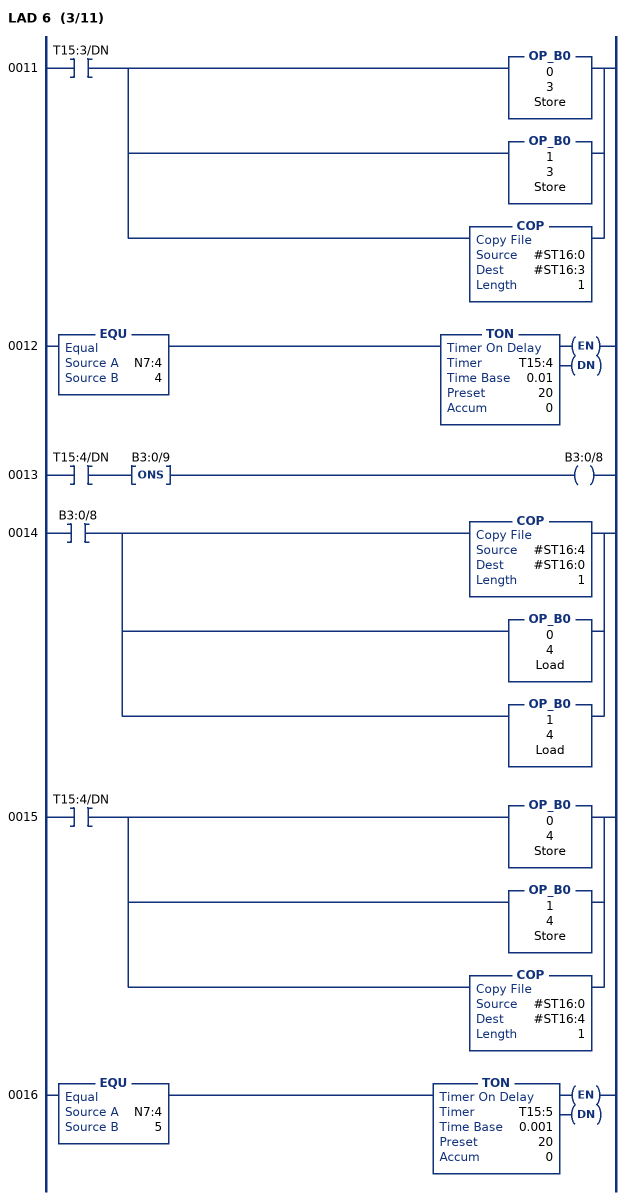
% Rung: 11 %
SOR XIC T15:3/DN BST OP_B0 0 3 Store NXB OP_B0 1 3 Store NXB COP #ST16:0 #ST16:3 1 BND EOR
% Rung: 12 %
SOR EQU N7:4 4 TON T15:4 0.01 20 0 EOR
% Rung: 13 %
SOR XIC T15:4/DN ONS B3:0/9 OTE B3:0/8 EOR
% Rung: 14 %
SOR XIC B3:0/8 BST COP #ST16:4 #ST16:0 1 NXB OP_B0 0 4 Load NXB OP_B0 1 4 Load BND EOR
% Rung: 15 %
SOR XIC T15:4/DN BST OP_B0 0 4 Store NXB OP_B0 1 4 Store NXB COP #ST16:0 #ST16:4 1 BND EOR
% Rung: 16 %
SOR EQU N7:4 5 TON T15:5 0.001 20 0 EOR

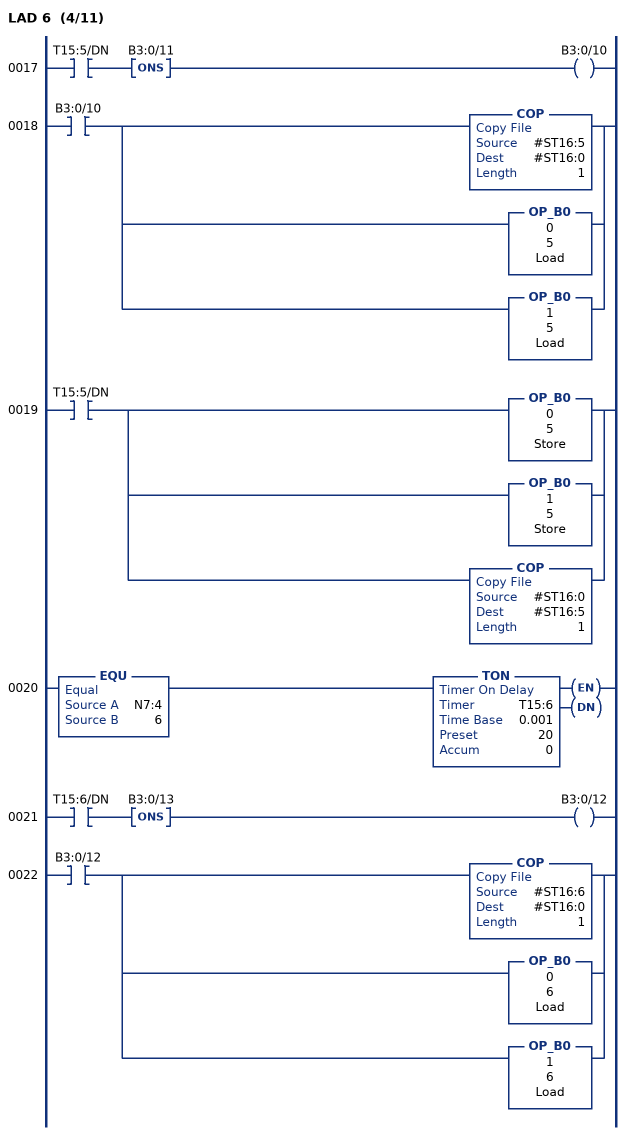
% Rung: 17 %
SOR XIC T15:5/DN ONS B3:0/11 OTE B3:0/10 EOR
% Rung: 18 %
SOR XIC B3:0/10 BST COP #ST16:5 #ST16:0 1 NXB OP_B0 0 5 Load NXB OP_B0 1 5 Load BND EOR
% Rung: 19 %
SOR XIC T15:5/DN BST OP_B0 0 5 Store NXB OP_B0 1 5 Store NXB COP #ST16:0 #ST16:5 1 BND EOR
% Rung: 20 %
SOR EQU N7:4 6 TON T15:6 0.001 20 0 EOR
% Rung: 21 %
SOR XIC T15:6/DN ONS B3:0/13 OTE B3:0/12 EOR
% Rung: 22 %
SOR XIC B3:0/12 BST COP #ST16:6 #ST16:0 1 NXB OP_B0 0 6 Load NXB OP_B0 1 6 Load BND EOR

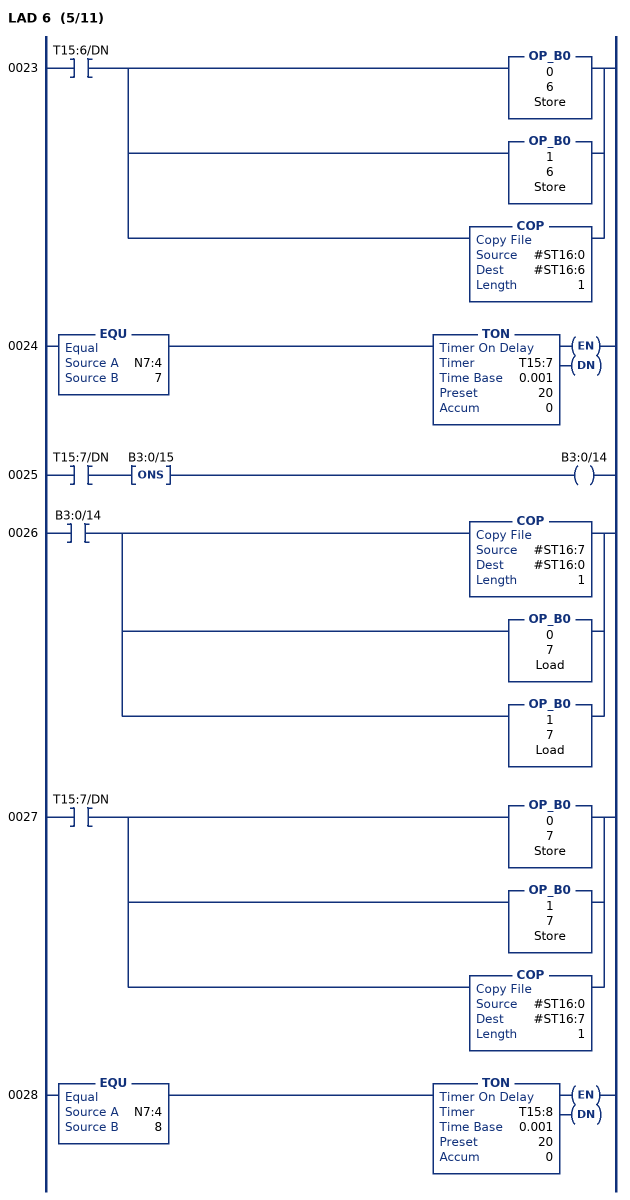
% Rung: 23 %
SOR XIC T15:6/DN BST OP_B0 0 6 Store NXB OP_B0 1 6 Store NXB COP #ST16:0 #ST16:6 1 BND EOR
% Rung: 24 %
SOR EQU N7:4 7 TON T15:7 0.001 20 0 EOR
% Rung: 25 %
SOR XIC T15:7/DN ONS B3:0/15 OTE B3:0/14 EOR
% Rung: 26 %
SOR XIC B3:0/14 BST COP #ST16:7 #ST16:0 1 NXB OP_B0 0 7 Load NXB OP_B0 1 7 Load BND EOR
% Rung: 27 %
SOR XIC T15:7/DN BST OP_B0 0 7 Store NXB OP_B0 1 7 Store NXB COP #ST16:0 #ST16:7 1 BND EOR
% Rung: 28 %
SOR EQU N7:4 8 TON T15:8 0.001 20 0 EOR

